    GP1:
        UF : 6, UT : 5,     CONFIG: 'N U T, 0, 0, 0',
       X = -410.7 mm, Y = 413.9 mm, Z = 598.9 mm,
       W = -11.9 deg, P = 9.7 deg,
    GP2:
        UF : 1, UT : 2,
       J1 = 0.0 deg, J2 = 0.0 deg
 };
P[387] {
    GP1:
        UF : 6, UT : 5,     CONFIG: 'N U T, 0, 0, 0',
 X = -393.7 mm, Y = 484.9 mm, Z = 598.9 mm,       W = -11.9 deg, P = 9.7 deg,
    GP2:
        UF : 1, UT : 2,
       J1 = 0.0 deg, J2 = 0.0 deg
 };
P[143] {
    GP1:
        UF : 6, UT : 5,     CONFIG: 'N U T, 0, 0, 0',
       X = -412.1 mm, Y = 415.1 mm, Z = 598.9 mm,
       W = -12.0 deg, P = 9.6 deg,
    GP2:
        UF : 1, UT : 2,
       J1 = 0.0 deg, J2 = 0.0 deg
 };
P[388] {
    GP1:
        UF : 6, UT : 5,     CONFIG: 'N U T, 0, 0, 0',
 X = -395.1 mm, Y = 486.1 mm, Z = 598.9 mm,       W = -12.0 deg, P = 9.6 deg,
    GP2:
        UF : 1, UT : 2,
       J1 = 0.0 deg, J2 = 0.0 deg
 };
P[144] {
    GP1:
        UF : 6, UT : 5,     CONFIG: 'N U T, 0, 0, 0',
       X = -413.0 mm, Y = 415.8 mm, Z = 598.9 mm,
       W = -11.9 deg, P = 9.6 deg,
    GP2:
        UF : 1, UT : 2,
       J1 = 0.0 deg, J2 = 0.0 deg
 };
P[389] {
    GP1:
        UF : 6, UT : 5,     CONFIG: 'N U T, 0, 0, 0',
 X = -396.0 mm, Y = 486.8 mm, Z = 598.9 mm,       W = -11.9 deg, P = 9.6 deg,
    GP2:
        UF : 1, UT : 2,
       J1 = 0.0 deg, J2 = 0.0 deg
 };
P[145] {
    GP1:
        UF : 6, UT : 5,     CONFIG: 'N U T, 0, 0, 0',
       X = -413.8 mm, Y = 416.5 mm, Z = 598.9 mm,
       W = -11.5 deg, P = 10.2 deg,
    GP2:
        UF : 1, UT : 2,
       J1 = 0.0 deg, J2 = 0.0 deg
 };
P[390] {
    GP1:
        UF : 6, UT : 5,     CONFIG: 'N U T, 0, 0, 0',
 X = -396.8 mm, Y = 487.5 mm, Z = 598.9 mm,       W = -11.5 deg, P = 10.2 deg,
    GP2:
        UF : 1, UT : 2,
       J1 = 0.0 deg, J2 = 0.0 deg
 };
P[146] {
    GP1:
        UF : 6, UT : 5,     CONFIG: 'N U T, 0, 0, 0',
       X = -414.8 mm, Y = 417.4 mm, Z = 598.9 mm,
       W = -11.4 deg, P = 10.5 deg,
    GP2:
        UF : 1, UT : 2,
       J1 = 0.0 deg, J2 = 0.0 deg
 };
P[391] {
    GP1:
        UF : 6, UT : 5,     CONFIG: 'N U T, 0, 0, 0',
 X = -397.8 mm, Y = 488.4 mm, Z = 598.9 mm,       W = -11.4 deg, P = 10.5 deg,
    GP2:
        UF : 1, UT : 2,
       J1 = 0.0 deg, J2 = 0.0 deg
 };
P[147] {
    GP1:
        UF : 6, UT : 5,     CONFIG: 'N U T, 0, 0, 0',
       X = -415.4 mm, Y = 417.9 mm, Z = 598.9 mm,
       W = -11.3 deg, P = 10.9 deg,
    GP2:
        UF : 1, UT : 2,
       J1 = 0.0 deg, J2 = 0.0 deg
 };
P[392] {
    GP1:
        UF : 6, UT : 5,     CONFIG: 'N U T, 0, 0, 0',
 X = -398.4 mm, Y = 488.9 mm, Z = 598.9 mm,       W = -11.3 deg, P = 10.9 deg,
    GP2:
        UF : 1, UT : 2,
       J1 = 0.0 deg, J2 = 0.0 deg
 };
P[148] {
    GP1:
        UF : 6, UT : 5,     CONFIG: 'N U T, 0, 0, 0',
       X = -415.8 mm, Y = 418.3 mm, Z = 598.9 mm,
       W = -10.8 deg, P = 11.6 deg,
    GP2:
        UF : 1, UT : 2,
       J1 = 0.0 deg, J2 = 0.0 deg
 };
P[393] {
    GP1:
        UF : 6, UT : 5,     CONFIG: 'N U T, 0, 0, 0',
 X = -398.8 mm, Y = 489.3 mm, Z = 598.9 mm,       W = -10.8 deg, P = 11.6 deg,
    GP2:
        UF : 1, UT : 2,
       J1 = 0.0 deg, J2 = 0.0 deg
 };
P[149] {
    GP1:
        UF : 6, UT : 5,     CONFIG: 'N U T, 0, 0, 0',
       X = -416.1 mm, Y = 418.7 mm, Z = 598.9 mm,
       W = -10.1 deg, P = 12.3 deg,
    GP2:
        UF : 1, UT : 2,
       J1 = 0.0 deg, J2 = 0.0 deg
 };
P[394] {
    GP1:
        UF : 6, UT : 5,     CONFIG: 'N U T, 0, 0, 0',
 X = -399.1 mm, Y = 489.7 mm, Z = 598.9 mm,       W = -10.1 deg, P = 12.3 deg,
    GP2:
        UF : 1, UT : 2,
       J1 = 0.0 deg, J2 = 0.0 deg
 };
P[150] {
    GP1:
        UF : 6, UT : 5,     CONFIG: 'N U T, 0, 0, 0',
       X = -416.8 mm, Y = 419.6 mm, Z = 598.9 mm,
       W = -9.7 deg, P = 12.7 deg,
    GP2:
        UF : 1, UT : 2,
       J1 = 0.0 deg, J2 = 0.0 deg
 };
P[395] {
    GP1:
        UF : 6, UT : 5,     CONFIG: 'N U T, 0, 0, 0',
 X = -399.8 mm, Y = 490.6 mm, Z = 598.9 mm,       W = -9.7 deg, P = 12.7 deg,
    GP2:
        UF : 1, UT : 2,
       J1 = 0.0 deg, J2 = 0.0 deg
 };
P[151] {
    GP1:
        UF : 6, UT : 5,     CONFIG: 'N U T, 0, 0, 0',
       X = -417.3 mm, Y = 420.2 mm, Z = 598.9 mm,
       W = -9.6 deg, P = 12.8 deg,
    GP2:
        UF : 1, UT : 2,
       J1 = 0.0 deg, J2 = 0.0 deg
 };
P[396] {
    GP1:
        UF : 6, UT : 5,     CONFIG: 'N U T, 0, 0, 0',
 X = -400.3 mm, Y = 491.2 mm, Z = 598.9 mm,       W = -9.6 deg, P = 12.8 deg,
    GP2:
        UF : 1, UT : 2,
       J1 = 0.0 deg, J2 = 0.0 deg
 };
P[152] {
    GP1:
        UF : 6, UT : 5,     CONFIG: 'N U T, 0, 0, 0',
       X = -417.9 mm, Y = 421.0 mm, Z = 598.9 mm,
       W = -8.6 deg, P = 13.4 deg,
    GP2:
        UF : 1, UT : 2,
       J1 = 0.0 deg, J2 = 0.0 deg
 };
P[397] {
    GP1:
        UF : 6, UT : 5,     CONFIG: 'N U T, 0, 0, 0',
 X = -400.9 mm, Y = 492.0 mm, Z = 598.9 mm,       W = -8.6 deg, P = 13.4 deg,
    GP2:
        UF : 1, UT : 2,
       J1 = 0.0 deg, J2 = 0.0 deg
 };
P[153] {
    GP1:
        UF : 6, UT : 5,     CONFIG: 'N U T, 0, 0, 0',
       X = -418.3 mm, Y = 421.8 mm, Z = 598.9 mm,
       W = -7.8 deg, P = 13.9 deg,
    GP2:
        UF : 1, UT : 2,
       J1 = 0.0 deg, J2 = 0.0 deg
 };
P[398] {
    GP1:
        UF : 6, UT : 5,     CONFIG: 'N U T, 0, 0, 0',
 X = -401.3 mm, Y = 492.8 mm, Z = 598.9 mm,       W = -7.8 deg, P = 13.9 deg,
    GP2:
        UF : 1, UT : 2,
       J1 = 0.0 deg, J2 = 0.0 deg
 };
P[154] {
    GP1:
        UF : 6, UT : 5,     CONFIG: 'N U T, 0, 0, 0',
       X = -418.8 mm, Y = 422.7 mm, Z = 598.9 mm,
       W = -7.5 deg, P = 13.9 deg,
    GP2:
        UF : 1, UT : 2,
       J1 = 0.0 deg, J2 = 0.0 deg
 };
P[399] {
    GP1:
        UF : 6, UT : 5,     CONFIG: 'N U T, 0, 0, 0',
 X = -401.8 mm, Y = 493.7 mm, Z = 598.9 mm,       W = -7.5 deg, P = 13.9 deg,
    GP2:
        UF : 1, UT : 2,
       J1 = 0.0 deg, J2 = 0.0 deg
 };
P[155] {
    GP1:
        UF : 6, UT : 5,     CONFIG: 'N U T, 0, 0, 0',
       X = -418.9 mm, Y = 423.0 mm, Z = 598.9 mm,
       W = -7.2 deg, P = 14.1 deg,
    GP2:
        UF : 1, UT : 2,
       J1 = 0.0 deg, J2 = 0.0 deg
 };
P[400] {
    GP1:
        UF : 6, UT : 5,     CONFIG: 'N U T, 0, 0, 0',
 X = -401.9 mm, Y = 494.0 mm, Z = 598.9 mm,       W = -7.2 deg, P = 14.1 deg,
    GP2:
        UF : 1, UT : 2,
       J1 = 0.0 deg, J2 = 0.0 deg
 };
P[156] {
    GP1:
        UF : 6, UT : 5,     CONFIG: 'N U T, 0, 0, 0',
       X = -419.0 mm, Y = 423.2 mm, Z = 598.9 mm,
       W = -6.9 deg, P = 14.2 deg,
    GP2:
        UF : 1, UT : 2,
       J1 = 0.0 deg, J2 = 0.0 deg
 };
P[401] {
    GP1:
        UF : 6, UT : 5,     CONFIG: 'N U T, 0, 0, 0',
 X = -402.0 mm, Y = 494.2 mm, Z = 598.9 mm,       W = -6.9 deg, P = 14.2 deg,
    GP2:
        UF : 1, UT : 2,
       J1 = 0.0 deg, J2 = 0.0 deg
 };
P[157] {
    GP1:
        UF : 6, UT : 5,     CONFIG: 'N U T, 0, 0, 0',
       X = -419.1 mm, Y = 423.4 mm, Z = 598.9 mm,
       W = -6.6 deg, P = 14.3 deg,
    GP2:
        UF : 1, UT : 2,
       J1 = 0.0 deg, J2 = 0.0 deg
 };
P[402] {
    GP1:
        UF : 6, UT : 5,     CONFIG: 'N U T, 0, 0, 0',
 X = -402.1 mm, Y = 494.4 mm, Z = 598.9 mm,       W = -6.6 deg, P = 14.3 deg,
    GP2:
        UF : 1, UT : 2,
       J1 = 0.0 deg, J2 = 0.0 deg
 };
P[158] {
    GP1:
        UF : 6, UT : 5,     CONFIG: 'N U T, 0, 0, 0',
       X = -419.3 mm, Y = 423.7 mm, Z = 598.9 mm,
       W = -6.3 deg, P = 14.4 deg,
    GP2:
        UF : 1, UT : 2,
       J1 = 0.0 deg, J2 = 0.0 deg
 };
P[403] {
    GP1:
        UF : 6, UT : 5,     CONFIG: 'N U T, 0, 0, 0',
 X = -402.3 mm, Y = 494.7 mm, Z = 598.9 mm,       W = -6.3 deg, P = 14.4 deg,
    GP2:
        UF : 1, UT : 2,
       J1 = 0.0 deg, J2 = 0.0 deg
 };
P[159] {
    GP1:
        UF : 6, UT : 5,     CONFIG: 'N U T, 0, 0, 0',
       X = -419.4 mm, Y = 424.0 mm, Z = 598.9 mm,
       W = -5.9 deg, P = 14.5 deg,
    GP2:
        UF : 1, UT : 2,
       J1 = 0.0 deg, J2 = 0.0 deg
 };
P[404] {
    GP1:
        UF : 6, UT : 5,     CONFIG: 'N U T, 0, 0, 0',
 X = -402.4 mm, Y = 495.0 mm, Z = 598.9 mm,       W = -5.9 deg, P = 14.5 deg,
    GP2:
        UF : 1, UT : 2,
       J1 = 0.0 deg, J2 = 0.0 deg
 };
P[160] {
    GP1:
        UF : 6, UT : 5,     CONFIG: 'N U T, 0, 0, 0',
       X = -419.5 mm, Y = 424.3 mm, Z = 598.9 mm,
       W = -5.6 deg, P = 14.5 deg,
    GP2:
        UF : 1, UT : 2,
       J1 = 0.0 deg, J2 = 0.0 deg
 };
P[405] {
    GP1:
        UF : 6, UT : 5,     CONFIG: 'N U T, 0, 0, 0',
 X = -402.5 mm, Y = 495.3 mm, Z = 598.9 mm,       W = -5.6 deg, P = 14.5 deg,
    GP2:
        UF : 1, UT : 2,
       J1 = 0.0 deg, J2 = 0.0 deg
 };
P[161] {
    GP1:
        UF : 6, UT : 5,     CONFIG: 'N U T, 0, 0, 0',
       X = -419.6 mm, Y = 424.6 mm, Z = 598.9 mm,
       W = -5.3 deg, P = 14.5 deg,
    GP2:
        UF : 1, UT : 2,
       J1 = 0.0 deg, J2 = 0.0 deg
 };
P[406] {
    GP1:
        UF : 6, UT : 5,     CONFIG: 'N U T, 0, 0, 0',
 X = -402.6 mm, Y = 495.6 mm, Z = 598.9 mm,       W = -5.3 deg, P = 14.5 deg,
    GP2:
        UF : 1, UT : 2,
       J1 = 0.0 deg, J2 = 0.0 deg
 };
P[162] {
    GP1:
        UF : 6, UT : 5,     CONFIG: 'N U T, 0, 0, 0',
       X = -419.7 mm, Y = 424.9 mm, Z = 598.9 mm,
       W = -4.9 deg, P = 14.6 deg,
    GP2:
        UF : 1, UT : 2,
       J1 = 0.0 deg, J2 = 0.0 deg
 };
P[407] {
    GP1:
        UF : 6, UT : 5,     CONFIG: 'N U T, 0, 0, 0',
 X = -402.7 mm, Y = 495.9 mm, Z = 598.9 mm,       W = -4.9 deg, P = 14.6 deg,
    GP2:
        UF : 1, UT : 2,
       J1 = 0.0 deg, J2 = 0.0 deg
 };
P[163] {
    GP1:
        UF : 6, UT : 5,     CONFIG: 'N U T, 0, 0, 0',
       X = -420.1 mm, Y = 426.4 mm, Z = 598.9 mm,
       W = -4.0 deg, P = 14.2 deg,
    GP2:
        UF : 1, UT : 2,
       J1 = 0.0 deg, J2 = 0.0 deg
 };
P[408] {
    GP1:
        UF : 6, UT : 5,     CONFIG: 'N U T, 0, 0, 0',
 X = -403.1 mm, Y = 497.4 mm, Z = 598.9 mm,       W = -4.0 deg, P = 14.2 deg,
    GP2:
        UF : 1, UT : 2,
       J1 = 0.0 deg, J2 = 0.0 deg
 };
P[164] {
    GP1:
        UF : 6, UT : 5,     CONFIG: 'N U T, 0, 0, 0',
       X = -420.2 mm, Y = 426.8 mm, Z = 598.9 mm,
       W = -3.4 deg, P = 14.2 deg,
    GP2:
        UF : 1, UT : 2,
       J1 = 0.0 deg, J2 = 0.0 deg
 };
P[409] {
    GP1:
        UF : 6, UT : 5,     CONFIG: 'N U T, 0, 0, 0',
 X = -403.2 mm, Y = 497.8 mm, Z = 598.9 mm,       W = -3.4 deg, P = 14.2 deg,
    GP2:
        UF : 1, UT : 2,
       J1 = 0.0 deg, J2 = 0.0 deg
 };
P[165] {
    GP1:
        UF : 6, UT : 5,     CONFIG: 'N U T, 0, 0, 0',
       X = -420.3 mm, Y = 427.0 mm, Z = 598.9 mm,
       W = -3.1 deg, P = 14.2 deg,
    GP2:
        UF : 1, UT : 2,
       J1 = 0.0 deg, J2 = 0.0 deg
 };
P[410] {
    GP1:
        UF : 6, UT : 5,     CONFIG: 'N U T, 0, 0, 0',
 X = -403.3 mm, Y = 498.0 mm, Z = 598.9 mm,       W = -3.1 deg, P = 14.2 deg,
    GP2:
        UF : 1, UT : 2,
       J1 = 0.0 deg, J2 = 0.0 deg
 };
P[166] {
    GP1:
        UF : 6, UT : 5,     CONFIG: 'N U T, 0, 0, 0',
       X = -420.4 mm, Y = 427.2 mm, Z = 598.9 mm,
       W = -2.8 deg, P = 14.2 deg,
    GP2:
        UF : 1, UT : 2,
       J1 = 0.0 deg, J2 = 0.0 deg
 };
P[411] {
    GP1:
        UF : 6, UT : 5,     CONFIG: 'N U T, 0, 0, 0',
 X = -403.4 mm, Y = 498.2 mm, Z = 598.9 mm,       W = -2.8 deg, P = 14.2 deg,
    GP2:
        UF : 1, UT : 2,
       J1 = 0.0 deg, J2 = 0.0 deg
 };
P[167] {
    GP1:
        UF : 6, UT : 5,     CONFIG: 'N U T, 0, 0, 0',
       X = -420.5 mm, Y = 428.0 mm, Z = 598.9 mm,
       W = -2.5 deg, P = 14.2 deg,
    GP2:
        UF : 1, UT : 2,
       J1 = 0.0 deg, J2 = 0.0 deg
 };
P[412] {
    GP1:
        UF : 6, UT : 5,     CONFIG: 'N U T, 0, 0, 0',
 X = -403.5 mm, Y = 499.0 mm, Z = 598.9 mm,       W = -2.5 deg, P = 14.2 deg,
    GP2:
        UF : 1, UT : 2,
       J1 = 0.0 deg, J2 = 0.0 deg
 };
P[168] {
    GP1:
        UF : 6, UT : 5,     CONFIG: 'N U T, 0, 0, 0',
       X = -420.7 mm, Y = 429.3 mm, Z = 598.9 mm,
       W = -1.5 deg, P = 14.1 deg,
    GP2:
        UF : 1, UT : 2,
       J1 = 0.0 deg, J2 = 0.0 deg
 };
P[413] {
    GP1:
        UF : 6, UT : 5,     CONFIG: 'N U T, 0, 0, 0',
 X = -403.7 mm, Y = 500.3 mm, Z = 598.9 mm,       W = -1.5 deg, P = 14.1 deg,
    GP2:
        UF : 1, UT : 2,
       J1 = 0.0 deg, J2 = 0.0 deg
 };
P[169] {
    GP1:
        UF : 6, UT : 5,     CONFIG: 'N U T, 0, 0, 0',
       X = -420.7 mm, Y = 429.7 mm, Z = 598.9 mm,
       W = -1.2 deg, P = 13.9 deg,
    GP2:
        UF : 1, UT : 2,
       J1 = 0.0 deg, J2 = 0.0 deg
 };
P[414] {
    GP1:
        UF : 6, UT : 5,     CONFIG: 'N U T, 0, 0, 0',
 X = -403.7 mm, Y = 500.7 mm, Z = 598.9 mm,       W = -1.2 deg, P = 13.9 deg,
    GP2:
        UF : 1, UT : 2,
       J1 = 0.0 deg, J2 = 0.0 deg
 };
P[170] {
    GP1:
        UF : 6, UT : 5,     CONFIG: 'N U T, 0, 0, 0',
       X = -420.7 mm, Y = 430.0 mm, Z = 598.9 mm,
       W = -0.8 deg, P = 13.6 deg,
    GP2:
        UF : 1, UT : 2,
       J1 = 0.0 deg, J2 = 0.0 deg
 };
P[415] {
    GP1:
        UF : 6, UT : 5,     CONFIG: 'N U T, 0, 0, 0',
 X = -403.7 mm, Y = 501.0 mm, Z = 598.9 mm,       W = -0.8 deg, P = 13.6 deg,
    GP2:
        UF : 1, UT : 2,
       J1 = 0.0 deg, J2 = 0.0 deg
 };
P[171] {
    GP1:
        UF : 6, UT : 5,     CONFIG: 'N U T, 0, 0, 0',
       X = -420.7 mm, Y = 430.4 mm, Z = 598.9 mm,
       W = -0.4 deg, P = 13.4 deg,
    GP2:
        UF : 1, UT : 2,
       J1 = 0.0 deg, J2 = 0.0 deg
 };
P[416] {
    GP1:
        UF : 6, UT : 5,     CONFIG: 'N U T, 0, 0, 0',
 X = -403.7 mm, Y = 501.4 mm, Z = 598.9 mm,       W = -0.4 deg, P = 13.4 deg,
    GP2:
        UF : 1, UT : 2,
       J1 = 0.0 deg, J2 = 0.0 deg
 };
P[172] {
    GP1:
        UF : 6, UT : 5,     CONFIG: 'N U T, 0, 0, 0',
       X = -420.7 mm, Y = 430.7 mm, Z = 598.9 mm,
       W = -0.1 deg, P = 13.2 deg,
    GP2:
        UF : 1, UT : 2,
       J1 = 0.0 deg, J2 = 0.0 deg
 };
P[417] {
    GP1:
        UF : 6, UT : 5,     CONFIG: 'N U T, 0, 0, 0',
 X = -403.7 mm, Y = 501.7 mm, Z = 598.9 mm,       W = -0.1 deg, P = 13.2 deg,
    GP2:
        UF : 1, UT : 2,
       J1 = 0.0 deg, J2 = 0.0 deg
 };
P[173] {
    GP1:
        UF : 6, UT : 5,     CONFIG: 'N U T, 0, 0, 0',
       X = -420.7 mm, Y = 432.1 mm, Z = 598.9 mm,
       W = 0.7 deg, P = 12.5 deg,
    GP2:
        UF : 1, UT : 2,
       J1 = 0.0 deg, J2 = 0.0 deg
 };
P[418] {
    GP1:
        UF : 6, UT : 5,     CONFIG: 'N U T, 0, 0, 0',
 X = -403.7 mm, Y = 503.1 mm, Z = 598.9 mm,       W = 0.7 deg, P = 12.5 deg,
    GP2:
        UF : 1, UT : 2,
       J1 = 0.0 deg, J2 = 0.0 deg
 };
P[174] {
    GP1:
        UF : 6, UT : 5,     CONFIG: 'N U T, 0, 0, 0',
       X = -420.7 mm, Y = 432.4 mm, Z = 598.9 mm,
       W = 0.9 deg, P = 12.3 deg,
    GP2:
        UF : 1, UT : 2,
       J1 = 0.0 deg, J2 = 0.0 deg
 };
P[419] {
    GP1:
        UF : 6, UT : 5,     CONFIG: 'N U T, 0, 0, 0',
 X = -403.7 mm, Y = 503.4 mm, Z = 598.9 mm,       W = 0.9 deg, P = 12.3 deg,
    GP2:
        UF : 1, UT : 2,
       J1 = 0.0 deg, J2 = 0.0 deg
 };
P[175] {
    GP1:
        UF : 6, UT : 5,     CONFIG: 'N U T, 0, 0, 0',
       X = -420.7 mm, Y = 432.7 mm, Z = 598.9 mm,
       W = 1.2 deg, P = 12.0 deg,
    GP2:
        UF : 1, UT : 2,
       J1 = 0.0 deg, J2 = 0.0 deg
 };
P[420] {
    GP1:
        UF : 6, UT : 5,     CONFIG: 'N U T, 0, 0, 0',
 X = -403.7 mm, Y = 503.7 mm, Z = 598.9 mm,       W = 1.2 deg, P = 12.0 deg,
    GP2:
        UF : 1, UT : 2,
       J1 = 0.0 deg, J2 = 0.0 deg
 };
P[176] {
    GP1:
        UF : 6, UT : 5,     CONFIG: 'N U T, 0, 0, 0',
       X = -420.6 mm, Y = 433.0 mm, Z = 598.9 mm,
       W = 1.4 deg, P = 11.8 deg,
    GP2:
        UF : 1, UT : 2,
       J1 = 0.0 deg, J2 = 0.0 deg
 };
P[421] {
    GP1:
        UF : 6, UT : 5,     CONFIG: 'N U T, 0, 0, 0',
 X = -403.6 mm, Y = 504.0 mm, Z = 598.9 mm,       W = 1.4 deg, P = 11.8 deg,
    GP2:
        UF : 1, UT : 2,
       J1 = 0.0 deg, J2 = 0.0 deg
 };
P[177] {
    GP1:
        UF : 6, UT : 5,     CONFIG: 'N U T, 0, 0, 0',
       X = -420.6 mm, Y = 433.4 mm, Z = 598.9 mm,
       W = 1.7 deg, P = 11.5 deg,
    GP2:
        UF : 1, UT : 2,
       J1 = 0.0 deg, J2 = 0.0 deg
 };
P[422] {
    GP1:
        UF : 6, UT : 5,     CONFIG: 'N U T, 0, 0, 0',
 X = -403.6 mm, Y = 504.4 mm, Z = 598.9 mm,       W = 1.7 deg, P = 11.5 deg,
    GP2:
        UF : 1, UT : 2,
       J1 = 0.0 deg, J2 = 0.0 deg
 };
P[178] {
    GP1:
        UF : 6, UT : 5,     CONFIG: 'N U T, 0, 0, 0',
       X = -420.3 mm, Y = 434.9 mm, Z = 598.9 mm,
       W = 2.3 deg, P = 11.3 deg,
    GP2:
        UF : 1, UT : 2,
       J1 = 0.0 deg, J2 = 0.0 deg
 };
P[423] {
    GP1:
        UF : 6, UT : 5,     CONFIG: 'N U T, 0, 0, 0',
 X = -403.3 mm, Y = 505.9 mm, Z = 598.9 mm,       W = 2.3 deg, P = 11.3 deg,
    GP2:
        UF : 1, UT : 2,
       J1 = 0.0 deg, J2 = 0.0 deg
 };
P[179] {
    GP1:
        UF : 6, UT : 5,     CONFIG: 'N U T, 0, 0, 0',
       X = -420.1 mm, Y = 435.7 mm, Z = 598.9 mm,
       W = 3.0 deg, P = 10.9 deg,
    GP2:
        UF : 1, UT : 2,
       J1 = 0.0 deg, J2 = 0.0 deg
 };
P[424] {
    GP1:
        UF : 6, UT : 5,     CONFIG: 'N U T, 0, 0, 0',
 X = -403.1 mm, Y = 506.7 mm, Z = 598.9 mm,       W = 3.0 deg, P = 10.9 deg,
    GP2:
        UF : 1, UT : 2,
       J1 = 0.0 deg, J2 = 0.0 deg
 };
P[180] {
    GP1:
        UF : 6, UT : 5,     CONFIG: 'N U T, 0, 0, 0',
       X = -419.9 mm, Y = 436.5 mm, Z = 598.9 mm,
       W = 3.4 deg, P = 9.7 deg,
    GP2:
        UF : 1, UT : 2,
       J1 = 0.0 deg, J2 = 0.0 deg
 };
P[425] {
    GP1:
        UF : 6, UT : 5,     CONFIG: 'N U T, 0, 0, 0',
 X = -402.9 mm, Y = 507.5 mm, Z = 598.9 mm,       W = 3.4 deg, P = 9.7 deg,
    GP2:
        UF : 1, UT : 2,
       J1 = 0.0 deg, J2 = 0.0 deg
 };
P[181] {
    GP1:
        UF : 6, UT : 5,     CONFIG: 'N U T, 0, 0, 0',
       X = -419.6 mm, Y = 437.3 mm, Z = 598.9 mm,
       W = 3.3 deg, P = 9.1 deg,
    GP2:
        UF : 1, UT : 2,
       J1 = 0.0 deg, J2 = 0.0 deg
 };
P[426] {
    GP1:
        UF : 6, UT : 5,     CONFIG: 'N U T, 0, 0, 0',
 X = -402.6 mm, Y = 508.3 mm, Z = 598.9 mm,       W = 3.3 deg, P = 9.1 deg,
    GP2:
        UF : 1, UT : 2,
       J1 = 0.0 deg, J2 = 0.0 deg
 };
P[182] {
    GP1:
        UF : 6, UT : 5,     CONFIG: 'N U T, 0, 0, 0',
       X = -419.2 mm, Y = 438.2 mm, Z = 598.9 mm,
       W = 3.7 deg, P = 8.7 deg,
    GP2:
        UF : 1, UT : 2,
       J1 = 0.0 deg, J2 = 0.0 deg
 };
P[427] {
    GP1:
        UF : 6, UT : 5,     CONFIG: 'N U T, 0, 0, 0',
 X = -402.2 mm, Y = 509.2 mm, Z = 598.9 mm,       W = 3.7 deg, P = 8.7 deg,
    GP2:
        UF : 1, UT : 2,
       J1 = 0.0 deg, J2 = 0.0 deg
 };
P[183] {
    GP1:
        UF : 6, UT : 5,     CONFIG: 'N U T, 0, 0, 0',
       X = -419.1 mm, Y = 438.5 mm, Z = 598.9 mm,
       W = 3.8 deg, P = 8.4 deg,
    GP2:
        UF : 1, UT : 2,
       J1 = 0.0 deg, J2 = 0.0 deg
 };
P[428] {
    GP1:
        UF : 6, UT : 5,     CONFIG: 'N U T, 0, 0, 0',
 X = -402.1 mm, Y = 509.5 mm, Z = 598.9 mm,       W = 3.8 deg, P = 8.4 deg,
    GP2:
        UF : 1, UT : 2,
       J1 = 0.0 deg, J2 = 0.0 deg
 };
P[184] {
    GP1:
        UF : 6, UT : 5,     CONFIG: 'N U T, 0, 0, 0',
       X = -419.0 mm, Y = 438.7 mm, Z = 598.9 mm,
       W = 3.8 deg, P = 8.1 deg,
    GP2:
        UF : 1, UT : 2,
       J1 = 0.0 deg, J2 = 0.0 deg
 };
P[429] {
    GP1:
        UF : 6, UT : 5,     CONFIG: 'N U T, 0, 0, 0',
 X = -402.0 mm, Y = 509.7 mm, Z = 598.9 mm,       W = 3.8 deg, P = 8.1 deg,
    GP2:
        UF : 1, UT : 2,
       J1 = 0.0 deg, J2 = 0.0 deg
 };
P[185] {
    GP1:
        UF : 6, UT : 5,     CONFIG: 'N U T, 0, 0, 0',
       X = -418.9 mm, Y = 438.9 mm, Z = 598.9 mm,
       W = 3.9 deg, P = 7.9 deg,
    GP2:
        UF : 1, UT : 2,
       J1 = 0.0 deg, J2 = 0.0 deg
 };
P[430] {
    GP1:
        UF : 6, UT : 5,     CONFIG: 'N U T, 0, 0, 0',
 X = -401.9 mm, Y = 509.9 mm, Z = 598.9 mm,       W = 3.9 deg, P = 7.9 deg,
    GP2:
        UF : 1, UT : 2,
       J1 = 0.0 deg, J2 = 0.0 deg
 };
P[186] {
    GP1:
        UF : 6, UT : 5,     CONFIG: 'N U T, 0, 0, 0',
       X = -418.8 mm, Y = 439.2 mm, Z = 598.9 mm,
       W = 4.0 deg, P = 7.6 deg,
    GP2:
        UF : 1, UT : 2,
       J1 = 0.0 deg, J2 = 0.0 deg
 };
P[431] {
    GP1:
        UF : 6, UT : 5,     CONFIG: 'N U T, 0, 0, 0',
 X = -401.8 mm, Y = 510.2 mm, Z = 598.9 mm,       W = 4.0 deg, P = 7.6 deg,
    GP2:
        UF : 1, UT : 2,
       J1 = 0.0 deg, J2 = 0.0 deg
 };
P[187] {
    GP1:
        UF : 6, UT : 5,     CONFIG: 'N U T, 0, 0, 0',
       X = -418.1 mm, Y = 440.5 mm, Z = 598.9 mm,
       W = 3.5 deg, P = 6.0 deg,
    GP2:
        UF : 1, UT : 2,
       J1 = 0.0 deg, J2 = 0.0 deg
 };
P[432] {
    GP1:
        UF : 6, UT : 5,     CONFIG: 'N U T, 0, 0, 0',
 X = -401.1 mm, Y = 511.5 mm, Z = 598.9 mm,       W = 3.5 deg, P = 6.0 deg,
    GP2:
        UF : 1, UT : 2,
       J1 = 0.0 deg, J2 = 0.0 deg
 };
P[188] {
    GP1:
        UF : 6, UT : 5,     CONFIG: 'N U T, 0, 0, 0',
       X = -417.6 mm, Y = 441.3 mm, Z = 598.9 mm,
       W = 3.5 deg, P = 5.3 deg,
    GP2:
        UF : 1, UT : 2,
       J1 = 0.0 deg, J2 = 0.0 deg
 };
P[433] {
    GP1:
        UF : 6, UT : 5,     CONFIG: 'N U T, 0, 0, 0',
 X = -400.6 mm, Y = 512.3 mm, Z = 598.9 mm,       W = 3.5 deg, P = 5.3 deg,
    GP2:
        UF : 1, UT : 2,
       J1 = 0.0 deg, J2 = 0.0 deg
 };
P[189] {
    GP1:
        UF : 6, UT : 5,     CONFIG: 'N U T, 0, 0, 0',
       X = -417.5 mm, Y = 441.4 mm, Z = 598.9 mm,
       W = 3.5 deg, P = 5.1 deg,
    GP2:
        UF : 1, UT : 2,
       J1 = 0.0 deg, J2 = 0.0 deg
 };
P[434] {
    GP1:
        UF : 6, UT : 5,     CONFIG: 'N U T, 0, 0, 0',
 X = -400.5 mm, Y = 512.4 mm, Z = 598.9 mm,       W = 3.5 deg, P = 5.1 deg,
    GP2:
        UF : 1, UT : 2,
       J1 = 0.0 deg, J2 = 0.0 deg
 };
P[190] {
    GP1:
        UF : 6, UT : 5,     CONFIG: 'N U T, 0, 0, 0',
       X = -417.4 mm, Y = 441.6 mm, Z = 598.9 mm,
       W = 3.5 deg, P = 4.9 deg,
    GP2:
        UF : 1, UT : 2,
       J1 = 0.0 deg, J2 = 0.0 deg
 };
P[435] {
    GP1:
        UF : 6, UT : 5,     CONFIG: 'N U T, 0, 0, 0',
 X = -400.4 mm, Y = 512.6 mm, Z = 598.9 mm,       W = 3.5 deg, P = 4.9 deg,
    GP2:
        UF : 1, UT : 2,
       J1 = 0.0 deg, J2 = 0.0 deg
 };
P[191] {
    GP1:
        UF : 6, UT : 5,     CONFIG: 'N U T, 0, 0, 0',
       X = -417.3 mm, Y = 441.7 mm, Z = 598.9 mm,
       W = 3.5 deg, P = 4.8 deg,
    GP2:
        UF : 1, UT : 2,
       J1 = 0.0 deg, J2 = 0.0 deg
 };
P[436] {
    GP1:
        UF : 6, UT : 5,     CONFIG: 'N U T, 0, 0, 0',
 X = -400.3 mm, Y = 512.7 mm, Z = 598.9 mm,       W = 3.5 deg, P = 4.8 deg,
    GP2:
        UF : 1, UT : 2,
       J1 = 0.0 deg, J2 = 0.0 deg
 };
P[192] {
    GP1:
        UF : 6, UT : 5,     CONFIG: 'N U T, 0, 0, 0',
       X = -417.1 mm, Y = 441.9 mm, Z = 598.9 mm,
       W = 3.5 deg, P = 4.5 deg,
    GP2:
        UF : 1, UT : 2,
       J1 = 0.0 deg, J2 = 0.0 deg
 };
P[437] {
    GP1:
        UF : 6, UT : 5,     CONFIG: 'N U T, 0, 0, 0',
 X = -400.1 mm, Y = 512.9 mm, Z = 598.9 mm,       W = 3.5 deg, P = 4.5 deg,
    GP2:
        UF : 1, UT : 2,
       J1 = 0.0 deg, J2 = 0.0 deg
 };
P[193] {
    GP1:
        UF : 6, UT : 5,     CONFIG: 'N U T, 0, 0, 0',
       X = -416.6 mm, Y = 442.6 mm, Z = 598.9 mm,
       W = 3.2 deg, P = 4.0 deg,
    GP2:
        UF : 1, UT : 2,
       J1 = 0.0 deg, J2 = 0.0 deg
 };
P[438] {
    GP1:
        UF : 6, UT : 5,     CONFIG: 'N U T, 0, 0, 0',
 X = -399.6 mm, Y = 513.6 mm, Z = 598.9 mm,       W = 3.2 deg, P = 4.0 deg,
    GP2:
        UF : 1, UT : 2,
       J1 = 0.0 deg, J2 = 0.0 deg
 };
P[194] {
    GP1:
        UF : 6, UT : 5,     CONFIG: 'N U T, 0, 0, 0',
       X = -414.6 mm, Y = 444.9 mm, Z = 598.9 mm,
       W = 2.9 deg, P = 3.4 deg,
    GP2:
        UF : 1, UT : 2,
       J1 = 0.0 deg, J2 = 0.0 deg
 };
P[439] {
    GP1:
        UF : 6, UT : 5,     CONFIG: 'N U T, 0, 0, 0',
 X = -397.6 mm, Y = 515.9 mm, Z = 598.9 mm,       W = 2.9 deg, P = 3.4 deg,
    GP2:
        UF : 1, UT : 2,
       J1 = 0.0 deg, J2 = 0.0 deg
 };
P[195] {
    GP1:
        UF : 6, UT : 5,     CONFIG: 'N U T, 0, 0, 0',
       X = -407.9 mm, Y = 451.9 mm, Z = 598.9 mm,
       W = 2.8 deg, P = 3.2 deg,
    GP2:
        UF : 1, UT : 2,
       J1 = 0.0 deg, J2 = 0.0 deg
 };
P[440] {
    GP1:
        UF : 6, UT : 5,     CONFIG: 'N U T, 0, 0, 0',
 X = -390.9 mm, Y = 522.9 mm, Z = 598.9 mm,       W = 2.8 deg, P = 3.2 deg,
    GP2:
        UF : 1, UT : 2,
       J1 = 0.0 deg, J2 = 0.0 deg
 };
P[196] {
    GP1:
        UF : 6, UT : 5,     CONFIG: 'N U T, 0, 0, 0',
       X = -401.2 mm, Y = 458.8 mm, Z = 598.9 mm,
       W = 2.6 deg, P = 3.0 deg,
    GP2:
        UF : 1, UT : 2,
       J1 = 0.0 deg, J2 = 0.0 deg
 };
P[441] {
    GP1:
        UF : 6, UT : 5,     CONFIG: 'N U T, 0, 0, 0',
 X = -384.2 mm, Y = 529.8 mm, Z = 598.9 mm,       W = 2.6 deg, P = 3.0 deg,
    GP2:
        UF : 1, UT : 2,
       J1 = 0.0 deg, J2 = 0.0 deg
 };
P[197] {
    GP1:
        UF : 6, UT : 5,     CONFIG: 'N U T, 0, 0, 0',
       X = -394.3 mm, Y = 465.6 mm, Z = 598.9 mm,
       W = 2.4 deg, P = 2.8 deg,
    GP2:
        UF : 1, UT : 2,
       J1 = 0.0 deg, J2 = 0.0 deg
 };
P[442] {
    GP1:
        UF : 6, UT : 5,     CONFIG: 'N U T, 0, 0, 0',
 X = -377.3 mm, Y = 536.6 mm, Z = 598.9 mm,       W = 2.4 deg, P = 2.8 deg,
    GP2:
        UF : 1, UT : 2,
       J1 = 0.0 deg, J2 = 0.0 deg
 };
P[198] {
    GP1:
        UF : 6, UT : 5,     CONFIG: 'N U T, 0, 0, 0',
       X = -387.4 mm, Y = 472.3 mm, Z = 598.9 mm,
       W = 2.2 deg, P = 2.6 deg,
    GP2:
        UF : 1, UT : 2,
       J1 = 0.0 deg, J2 = 0.0 deg
 };
P[443] {
    GP1:
        UF : 6, UT : 5,     CONFIG: 'N U T, 0, 0, 0',
 X = -370.4 mm, Y = 543.3 mm, Z = 598.9 mm,       W = 2.2 deg, P = 2.6 deg,
    GP2:
        UF : 1, UT : 2,
       J1 = 0.0 deg, J2 = 0.0 deg
 };
P[199] {
    GP1:
        UF : 6, UT : 5,     CONFIG: 'N U T, 0, 0, 0',
       X = -383.7 mm, Y = 475.8 mm, Z = 598.9 mm,
       W = 2.1 deg, P = 2.5 deg,
    GP2:
        UF : 1, UT : 2,
       J1 = 0.0 deg, J2 = 0.0 deg
 };
P[444] {
    GP1:
        UF : 6, UT : 5,     CONFIG: 'N U T, 0, 0, 0',
 X = -366.7 mm, Y = 546.8 mm, Z = 598.9 mm,       W = 2.1 deg, P = 2.5 deg,
    GP2:
        UF : 1, UT : 2,
       J1 = 0.0 deg, J2 = 0.0 deg
 };
P[200] {
    GP1:
        UF : 6, UT : 5,     CONFIG: 'N U T, 0, 0, 0',
       X = -382.4 mm, Y = 477.2 mm, Z = 598.9 mm,
       W = 2.1 deg, P = 2.5 deg,
    GP2:
        UF : 1, UT : 2,
       J1 = 0.0 deg, J2 = 0.0 deg
 };
P[445] {
    GP1:
        UF : 6, UT : 5,     CONFIG: 'N U T, 0, 0, 0',
 X = -365.4 mm, Y = 548.2 mm, Z = 598.9 mm,       W = 2.1 deg, P = 2.5 deg,
    GP2:
        UF : 1, UT : 2,
       J1 = 0.0 deg, J2 = 0.0 deg
 };
P[201] {
    GP1:
        UF : 6, UT : 5,     CONFIG: 'N U T, 0, 0, 0',
       X = -381.1 mm, Y = 478.6 mm, Z = 598.9 mm,
       W = 2.1 deg, P = 2.4 deg,
    GP2:
        UF : 1, UT : 2,
       J1 = 0.0 deg, J2 = 0.0 deg
 };
P[446] {
    GP1:
        UF : 6, UT : 5,     CONFIG: 'N U T, 0, 0, 0',
 X = -364.1 mm, Y = 549.6 mm, Z = 598.9 mm,       W = 2.1 deg, P = 2.4 deg,
    GP2:
        UF : 1, UT : 2,
       J1 = 0.0 deg, J2 = 0.0 deg
 };
P[202] {
    GP1:
        UF : 6, UT : 5,     CONFIG: 'N U T, 0, 0, 0',
       X = -380.3 mm, Y = 479.6 mm, Z = 598.9 mm,
       W = 2.0 deg, P = 2.4 deg,
    GP2:
        UF : 1, UT : 2,
       J1 = 0.0 deg, J2 = 0.0 deg
 };
P[447] {
    GP1:
        UF : 6, UT : 5,     CONFIG: 'N U T, 0, 0, 0',
 X = -363.3 mm, Y = 550.6 mm, Z = 598.9 mm,       W = 2.0 deg, P = 2.4 deg,
    GP2:
        UF : 1, UT : 2,
       J1 = 0.0 deg, J2 = 0.0 deg
 };
P[203] {
    GP1:
        UF : 6, UT : 5,     CONFIG: 'N U T, 0, 0, 0',
       X = -379.7 mm, Y = 480.8 mm, Z = 598.9 mm,
       W = 2.0 deg, P = 2.4 deg,
    GP2:
        UF : 1, UT : 2,
       J1 = 0.0 deg, J2 = 0.0 deg
 };
P[448] {
    GP1:
        UF : 6, UT : 5,     CONFIG: 'N U T, 0, 0, 0',
 X = -362.7 mm, Y = 551.8 mm, Z = 598.9 mm,       W = 2.0 deg, P = 2.4 deg,
    GP2:
        UF : 1, UT : 2,
       J1 = 0.0 deg, J2 = 0.0 deg
 };
P[204] {
    GP1:
        UF : 6, UT : 5,     CONFIG: 'N U T, 0, 0, 0',
       X = -379.2 mm, Y = 482.0 mm, Z = 598.9 mm,
       W = 1.9 deg, P = 2.4 deg,
    GP2:
        UF : 1, UT : 2,
       J1 = 0.0 deg, J2 = 0.0 deg
 };
P[449] {
    GP1:
        UF : 6, UT : 5,     CONFIG: 'N U T, 0, 0, 0',
 X = -362.2 mm, Y = 553.0 mm, Z = 598.9 mm,       W = 1.9 deg, P = 2.4 deg,
    GP2:
        UF : 1, UT : 2,
       J1 = 0.0 deg, J2 = 0.0 deg
 };
P[205] {
    GP1:
        UF : 6, UT : 5,     CONFIG: 'N U T, 0, 0, 0',
       X = -378.7 mm, Y = 484.0 mm, Z = 598.9 mm,
       W = 1.9 deg, P = 2.3 deg,
    GP2:
        UF : 1, UT : 2,
       J1 = 0.0 deg, J2 = 0.0 deg
 };
P[450] {
    GP1:
        UF : 6, UT : 5,     CONFIG: 'N U T, 0, 0, 0',
 X = -361.7 mm, Y = 555.0 mm, Z = 598.9 mm,       W = 1.9 deg, P = 2.3 deg,
    GP2:
        UF : 1, UT : 2,
       J1 = 0.0 deg, J2 = 0.0 deg
 };
P[206] {
    GP1:
        UF : 6, UT : 5,     CONFIG: 'N U T, 0, 0, 0',
       X = -378.5 mm, Y = 486.3 mm, Z = 598.9 mm,
       W = 1.9 deg, P = 2.2 deg,
    GP2:
        UF : 1, UT : 2,
       J1 = 0.0 deg, J2 = 0.0 deg
 };
P[451] {
    GP1:
        UF : 6, UT : 5,     CONFIG: 'N U T, 0, 0, 0',
 X = -361.5 mm, Y = 557.3 mm, Z = 598.9 mm,       W = 1.9 deg, P = 2.2 deg,
    GP2:
        UF : 1, UT : 2,
       J1 = 0.0 deg, J2 = 0.0 deg
 };
P[207] {
    GP1:
        UF : 6, UT : 5,     CONFIG: 'N U T, 0, 0, 0',
       X = -378.7 mm, Y = 488.4 mm, Z = 598.9 mm,
       W = 1.8 deg, P = 2.2 deg,
    GP2:
        UF : 1, UT : 2,
       J1 = 0.0 deg, J2 = 0.0 deg
 };
P[452] {
    GP1:
        UF : 6, UT : 5,     CONFIG: 'N U T, 0, 0, 0',
 X = -361.7 mm, Y = 559.4 mm, Z = 598.9 mm,       W = 1.8 deg, P = 2.2 deg,
    GP2:
        UF : 1, UT : 2,
       J1 = 0.0 deg, J2 = 0.0 deg
 };
P[208] {
    GP1:
        UF : 6, UT : 5,     CONFIG: 'N U T, 0, 0, 0',
       X = -379.4 mm, Y = 490.6 mm, Z = 598.9 mm,
       W = 1.8 deg, P = 2.1 deg,
    GP2:
        UF : 1, UT : 2,
       J1 = 0.0 deg, J2 = 0.0 deg
 };
P[453] {
    GP1:
        UF : 6, UT : 5,     CONFIG: 'N U T, 0, 0, 0',
 X = -362.4 mm, Y = 561.6 mm, Z = 598.9 mm,       W = 1.8 deg, P = 2.1 deg,
    GP2:
        UF : 1, UT : 2,
       J1 = 0.0 deg, J2 = 0.0 deg
 };
P[209] {
    GP1:
        UF : 6, UT : 5,     CONFIG: 'N U T, 0, 0, 0',
       X = -380.0 mm, Y = 491.8 mm, Z = 598.9 mm,
       W = 1.8 deg, P = 2.1 deg,
    GP2:
        UF : 1, UT : 2,
       J1 = 0.0 deg, J2 = 0.0 deg
 };
P[454] {
    GP1:
        UF : 6, UT : 5,     CONFIG: 'N U T, 0, 0, 0',
 X = -363.0 mm, Y = 562.8 mm, Z = 598.9 mm,       W = 1.8 deg, P = 2.1 deg,
    GP2:
        UF : 1, UT : 2,
       J1 = 0.0 deg, J2 = 0.0 deg
 };
P[210] {
    GP1:
        UF : 6, UT : 5,     CONFIG: 'N U T, 0, 0, 0',
       X = -380.9 mm, Y = 492.9 mm, Z = 598.9 mm,
       W = 1.8 deg, P = 2.1 deg,
    GP2:
        UF : 1, UT : 2,
       J1 = 0.0 deg, J2 = 0.0 deg
 };
P[455] {
    GP1:
        UF : 6, UT : 5,     CONFIG: 'N U T, 0, 0, 0',
 X = -363.9 mm, Y = 563.9 mm, Z = 598.9 mm,       W = 1.8 deg, P = 2.1 deg,
    GP2:
        UF : 1, UT : 2,
       J1 = 0.0 deg, J2 = 0.0 deg
 };
P[211] {
    GP1:
        UF : 6, UT : 5,     CONFIG: 'N U T, 0, 0, 0',
       X = -382.0 mm, Y = 494.0 mm, Z = 598.9 mm,
       W = 1.7 deg, P = 2.1 deg,
    GP2:
        UF : 1, UT : 2,
       J1 = 0.0 deg, J2 = 0.0 deg
 };
P[456] {
    GP1:
        UF : 6, UT : 5,     CONFIG: 'N U T, 0, 0, 0',
 X = -365.0 mm, Y = 565.0 mm, Z = 598.9 mm,       W = 1.7 deg, P = 2.1 deg,
    GP2:
        UF : 1, UT : 2,
       J1 = 0.0 deg, J2 = 0.0 deg
 };
P[212] {
    GP1:
        UF : 6, UT : 5,     CONFIG: 'N U T, 0, 0, 0',
       X = -384.2 mm, Y = 495.8 mm, Z = 598.9 mm,
       W = 1.7 deg, P = 2.0 deg,
    GP2:
        UF : 1, UT : 2,
       J1 = 0.0 deg, J2 = 0.0 deg
 };
P[457] {
    GP1:
        UF : 6, UT : 5,     CONFIG: 'N U T, 0, 0, 0',
 X = -367.2 mm, Y = 566.8 mm, Z = 598.9 mm,       W = 1.7 deg, P = 2.0 deg,
    GP2:
        UF : 1, UT : 2,
       J1 = 0.0 deg, J2 = 0.0 deg
 };
P[213] {
    GP1:
        UF : 6, UT : 5,     CONFIG: 'N U T, 0, 0, 0',
       X = -392.3 mm, Y = 501.0 mm, Z = 598.9 mm,
       W = 1.5 deg, P = 1.8 deg,
    GP2:
        UF : 1, UT : 2,
       J1 = 0.0 deg, J2 = 0.0 deg
 };
P[458] {
    GP1:
        UF : 6, UT : 5,     CONFIG: 'N U T, 0, 0, 0',
 X = -375.3 mm, Y = 572.0 mm, Z = 598.9 mm,       W = 1.5 deg, P = 1.8 deg,
    GP2:
        UF : 1, UT : 2,
       J1 = 0.0 deg, J2 = 0.0 deg
 };
P[214] {
    GP1:
        UF : 6, UT : 5,     CONFIG: 'N U T, 0, 0, 0',
       X = -400.5 mm, Y = 506.1 mm, Z = 598.9 mm,
       W = 1.3 deg, P = 1.5 deg,
    GP2:
        UF : 1, UT : 2,
       J1 = 0.0 deg, J2 = 0.0 deg
 };
P[459] {
    GP1:
        UF : 6, UT : 5,     CONFIG: 'N U T, 0, 0, 0',
 X = -383.5 mm, Y = 577.1 mm, Z = 598.9 mm,       W = 1.3 deg, P = 1.5 deg,
    GP2:
        UF : 1, UT : 2,
       J1 = 0.0 deg, J2 = 0.0 deg
 };
P[215] {
    GP1:
        UF : 6, UT : 5,     CONFIG: 'N U T, 0, 0, 0',
       X = -408.8 mm, Y = 511.0 mm, Z = 598.9 mm,
       W = 1.1 deg, P = 1.3 deg,
    GP2:
        UF : 1, UT : 2,
       J1 = 0.0 deg, J2 = 0.0 deg
 };
P[460] {
    GP1:
        UF : 6, UT : 5,     CONFIG: 'N U T, 0, 0, 0',
 X = -391.8 mm, Y = 582.0 mm, Z = 598.9 mm,       W = 1.1 deg, P = 1.3 deg,
    GP2:
        UF : 1, UT : 2,
       J1 = 0.0 deg, J2 = 0.0 deg
 };
P[216] {
    GP1:
        UF : 6, UT : 5,     CONFIG: 'N U T, 0, 0, 0',
       X = -417.2 mm, Y = 515.8 mm, Z = 598.9 mm,
       W = 1.0 deg, P = 1.1 deg,
    GP2:
        UF : 1, UT : 2,
       J1 = 0.0 deg, J2 = 0.0 deg
 };
P[461] {
    GP1:
        UF : 6, UT : 5,     CONFIG: 'N U T, 0, 0, 0',
 X = -400.2 mm, Y = 586.8 mm, Z = 598.9 mm,       W = 1.0 deg, P = 1.1 deg,
    GP2:
        UF : 1, UT : 2,
       J1 = 0.0 deg, J2 = 0.0 deg
 };
P[217] {
    GP1:
        UF : 6, UT : 5,     CONFIG: 'N U T, 0, 0, 0',
       X = -425.6 mm, Y = 520.4 mm, Z = 598.9 mm,
       W = 0.8 deg, P = 0.9 deg,
    GP2:
        UF : 1, UT : 2,
       J1 = 0.0 deg, J2 = 0.0 deg
 };
P[462] {
    GP1:
        UF : 6, UT : 5,     CONFIG: 'N U T, 0, 0, 0',
 X = -408.6 mm, Y = 591.4 mm, Z = 598.9 mm,       W = 0.8 deg, P = 0.9 deg,
    GP2:
        UF : 1, UT : 2,
       J1 = 0.0 deg, J2 = 0.0 deg
 };
P[218] {
    GP1:
        UF : 6, UT : 5,     CONFIG: 'N U T, 0, 0, 0',
       X = -434.2 mm, Y = 524.9 mm, Z = 598.9 mm,
       W = 0.6 deg, P = 0.7 deg,
    GP2:
        UF : 1, UT : 2,
       J1 = 0.0 deg, J2 = 0.0 deg
 };
P[463] {
    GP1:
        UF : 6, UT : 5,     CONFIG: 'N U T, 0, 0, 0',
 X = -417.2 mm, Y = 595.9 mm, Z = 598.9 mm,       W = 0.6 deg, P = 0.7 deg,
    GP2:
        UF : 1, UT : 2,
       J1 = 0.0 deg, J2 = 0.0 deg
 };
P[219] {
    GP1:
        UF : 6, UT : 5,     CONFIG: 'N U T, 0, 0, 0',
       X = -439.8 mm, Y = 527.8 mm, Z = 598.9 mm,
       W = 0.5 deg, P = 0.6 deg,
    GP2:
        UF : 1, UT : 2,
       J1 = 0.0 deg, J2 = 0.0 deg
 };
P[464] {
    GP1:
        UF : 6, UT : 5,     CONFIG: 'N U T, 0, 0, 0',
 X = -422.8 mm, Y = 598.8 mm, Z = 598.9 mm,       W = 0.5 deg, P = 0.6 deg,
    GP2:
        UF : 1, UT : 2,
       J1 = 0.0 deg, J2 = 0.0 deg
 };
P[220] {
    GP1:
        UF : 6, UT : 5,     CONFIG: 'N U T, 0, 0, 0',
       X = -441.8 mm, Y = 528.9 mm, Z = 598.9 mm,
       W = 0.5 deg, P = 0.5 deg,
    GP2:
        UF : 1, UT : 2,
       J1 = 0.0 deg, J2 = 0.0 deg
 };
P[465] {
    GP1:
        UF : 6, UT : 5,     CONFIG: 'N U T, 0, 0, 0',
 X = -424.8 mm, Y = 599.9 mm, Z = 598.9 mm,       W = 0.5 deg, P = 0.5 deg,
    GP2:
        UF : 1, UT : 2,
       J1 = 0.0 deg, J2 = 0.0 deg
 };
P[221] {
    GP1:
        UF : 6, UT : 5,     CONFIG: 'N U T, 0, 0, 0',
       X = -443.4 mm, Y = 530.3 mm, Z = 598.9 mm,
       W = 0.4 deg, P = 0.5 deg,
    GP2:
        UF : 1, UT : 2,
       J1 = 0.0 deg, J2 = 0.0 deg
 };
P[466] {
    GP1:
        UF : 6, UT : 5,     CONFIG: 'N U T, 0, 0, 0',
 X = -426.4 mm, Y = 601.3 mm, Z = 598.9 mm,       W = 0.4 deg, P = 0.5 deg,
    GP2:
        UF : 1, UT : 2,
       J1 = 0.0 deg, J2 = 0.0 deg
 };
P[222] {
    GP1:
        UF : 6, UT : 5,     CONFIG: 'N U T, 0, 0, 0',
       X = -445.1 mm, Y = 531.9 mm, Z = 598.9 mm,
       W = 0.3 deg, P = 0.4 deg,
    GP2:
        UF : 1, UT : 2,
       J1 = 0.0 deg, J2 = 0.0 deg
 };
P[467] {
    GP1:
        UF : 6, UT : 5,     CONFIG: 'N U T, 0, 0, 0',
 X = -428.1 mm, Y = 602.9 mm, Z = 598.9 mm,       W = 0.3 deg, P = 0.4 deg,
    GP2:
        UF : 1, UT : 2,
       J1 = 0.0 deg, J2 = 0.0 deg
 };
P[223] {
    GP1:
        UF : 6, UT : 5,     CONFIG: 'N U T, 0, 0, 0',
       X = -446.2 mm, Y = 533.6 mm, Z = 598.9 mm,
       W = 0.3 deg, P = 0.4 deg,
    GP2:
        UF : 1, UT : 2,
       J1 = 0.0 deg, J2 = 0.0 deg
 };
P[468] {
    GP1:
        UF : 6, UT : 5,     CONFIG: 'N U T, 0, 0, 0',
 X = -429.2 mm, Y = 604.6 mm, Z = 598.9 mm,       W = 0.3 deg, P = 0.4 deg,
    GP2:
        UF : 1, UT : 2,
       J1 = 0.0 deg, J2 = 0.0 deg
 };
P[224] {
    GP1:
        UF : 6, UT : 5,     CONFIG: 'N U T, 0, 0, 0',
       X = -451.4 mm, Y = 542.1 mm, Z = 598.9 mm,
       W = 0.1 deg, P = 0.2 deg,
    GP2:
        UF : 1, UT : 2,
       J1 = 0.0 deg, J2 = 0.0 deg
 };
P[469] {
    GP1:
        UF : 6, UT : 5,     CONFIG: 'N U T, 0, 0, 0',
 X = -434.4 mm, Y = 613.1 mm, Z = 598.9 mm,       W = 0.1 deg, P = 0.2 deg,
    GP2:
        UF : 1, UT : 2,
       J1 = 0.0 deg, J2 = 0.0 deg
 };
P[225] {
    GP1:
        UF : 6, UT : 5,     CONFIG: 'N U T, 0, 0, 0',
       X = -456.5 mm, Y = 550.7 mm, Z = 598.9 mm,
       W = 0.0 deg, P = 0.0 deg,
    GP2:
        UF : 1, UT : 2,
       J1 = 0.0 deg, J2 = 0.0 deg
 };
P[470] {
    GP1:
        UF : 6, UT : 5,     CONFIG: 'N U T, 0, 0, 0',
 X = -439.5 mm, Y = 621.7 mm, Z = 598.9 mm,       W = 0.0 deg, P = 0.0 deg,
    GP2:
        UF : 1, UT : 2,
       J1 = 0.0 deg, J2 = 0.0 deg
 };
P[226] {
    GP1:
        UF : 6, UT : 5,     CONFIG: 'N U T, 0, 0, 0',
       X = -457.7 mm, Y = 552.8 mm, Z = 598.9 mm,
       W = 0.0 deg, P = 0.0 deg,
    GP2:
        UF : 1, UT : 2,
       J1 = 0.0 deg, J2 = 0.0 deg
 };
P[471] {
    GP1:
        UF : 6, UT : 5,     CONFIG: 'N U T, 0, 0, 0',
 X = -440.7 mm, Y = 623.8 mm, Z = 598.9 mm,       W = 0.0 deg, P = 0.0 deg,
    GP2:
        UF : 1, UT : 2,
       J1 = 0.0 deg, J2 = 0.0 deg
 };
P[227] {
    GP1:
        UF : 6, UT : 5,     CONFIG: 'N U T, 0, 0, 0',
       X = -458.1 mm, Y = 554.3 mm, Z = 598.9 mm,
       W = 0.0 deg, P = 0.0 deg,
    GP2:
        UF : 1, UT : 2,
       J1 = 0.0 deg, J2 = 0.0 deg
 };
P[472] {
    GP1:
        UF : 6, UT : 5,     CONFIG: 'N U T, 0, 0, 0',
 X = -441.1 mm, Y = 625.3 mm, Z = 598.9 mm,       W = 0.0 deg, P = 0.0 deg,
    GP2:
        UF : 1, UT : 2,
       J1 = 0.0 deg, J2 = 0.0 deg
 };
P[228] {
    GP1:
        UF : 6, UT : 5,     CONFIG: 'N U T, 0, 0, 0',
       X = -458.3 mm, Y = 555.2 mm, Z = 598.9 mm,
       W = 0.0 deg, P = 0.0 deg,
    GP2:
        UF : 1, UT : 2,
       J1 = 0.0 deg, J2 = 0.0 deg
 };
P[473] {
    GP1:
        UF : 6, UT : 5,     CONFIG: 'N U T, 0, 0, 0',
 X = -441.3 mm, Y = 626.2 mm, Z = 598.9 mm,       W = 0.0 deg, P = 0.0 deg,
    GP2:
        UF : 1, UT : 2,
       J1 = 0.0 deg, J2 = 0.0 deg
 };
P[229] {
    GP1:
        UF : 6, UT : 5,     CONFIG: 'N U T, 0, 0, 0',
       X = -458.3 mm, Y = 556.1 mm, Z = 598.9 mm,
       W = 0.0 deg, P = 0.0 deg,
    GP2:
        UF : 1, UT : 2,
       J1 = 0.0 deg, J2 = 0.0 deg
 };
P[474] {
    GP1:
        UF : 6, UT : 5,     CONFIG: 'N U T, 0, 0, 0',
 X = -441.3 mm, Y = 627.1 mm, Z = 598.9 mm,       W = 0.0 deg, P = 0.0 deg,
    GP2:
        UF : 1, UT : 2,
       J1 = 0.0 deg, J2 = 0.0 deg
 };
P[230] {
    GP1:
        UF : 6, UT : 5,     CONFIG: 'N U T, 0, 0, 0',
       X = -458.2 mm, Y = 557.0 mm, Z = 598.9 mm,
       W = 0.0 deg, P = 0.0 deg,
    GP2:
        UF : 1, UT : 2,
       J1 = 0.0 deg, J2 = 0.0 deg
 };
P[475] {
    GP1:
        UF : 6, UT : 5,     CONFIG: 'N U T, 0, 0, 0',
 X = -441.2 mm, Y = 628.0 mm, Z = 598.9 mm,       W = 0.0 deg, P = 0.0 deg,
    GP2:
        UF : 1, UT : 2,
       J1 = 0.0 deg, J2 = 0.0 deg
 };
P[231] {
    GP1:
        UF : 6, UT : 5,     CONFIG: 'N U T, 0, 0, 0',
       X = -457.8 mm, Y = 558.8 mm, Z = 598.9 mm,
       W = 0.0 deg, P = 0.0 deg,
    GP2:
        UF : 1, UT : 2,
       J1 = 0.0 deg, J2 = 0.0 deg
 };
P[476] {
    GP1:
        UF : 6, UT : 5,     CONFIG: 'N U T, 0, 0, 0',
 X = -440.8 mm, Y = 629.8 mm, Z = 598.9 mm,       W = 0.0 deg, P = 0.0 deg,
    GP2:
        UF : 1, UT : 2,
       J1 = 0.0 deg, J2 = 0.0 deg
 };
P[232] {
    GP1:
        UF : 6, UT : 5,     CONFIG: 'N U T, 0, 0, 0',
       X = -457.0 mm, Y = 560.3 mm, Z = 598.9 mm,
       W = 0.0 deg, P = 0.0 deg,
    GP2:
        UF : 1, UT : 2,
       J1 = 0.0 deg, J2 = 0.0 deg
 };
P[477] {
    GP1:
        UF : 6, UT : 5,     CONFIG: 'N U T, 0, 0, 0',
 X = -440.0 mm, Y = 631.3 mm, Z = 598.9 mm,       W = 0.0 deg, P = 0.0 deg,
    GP2:
        UF : 1, UT : 2,
       J1 = 0.0 deg, J2 = 0.0 deg
 };
P[233] {
    GP1:
        UF : 6, UT : 5,     CONFIG: 'N U T, 0, 0, 0',
       X = -455.9 mm, Y = 561.7 mm, Z = 598.9 mm,
       W = 0.0 deg, P = 0.0 deg,
    GP2:
        UF : 1, UT : 2,
       J1 = 0.0 deg, J2 = 0.0 deg
 };
P[478] {
    GP1:
        UF : 6, UT : 5,     CONFIG: 'N U T, 0, 0, 0',
 X = -438.9 mm, Y = 632.7 mm, Z = 598.9 mm,       W = 0.0 deg, P = 0.0 deg,
    GP2:
        UF : 1, UT : 2,
       J1 = 0.0 deg, J2 = 0.0 deg
 };
P[234] {
    GP1:
        UF : 6, UT : 5,     CONFIG: 'N U T, 0, 0, 0',
       X = -454.5 mm, Y = 562.8 mm, Z = 598.9 mm,
       W = 0.0 deg, P = 0.0 deg,
    GP2:
        UF : 1, UT : 2,
       J1 = 0.0 deg, J2 = 0.0 deg
 };
P[479] {
    GP1:
        UF : 6, UT : 5,     CONFIG: 'N U T, 0, 0, 0',
 X = -437.5 mm, Y = 633.8 mm, Z = 598.9 mm,       W = 0.0 deg, P = 0.0 deg,
    GP2:
        UF : 1, UT : 2,
       J1 = 0.0 deg, J2 = 0.0 deg
 };
P[235] {
    GP1:
        UF : 6, UT : 5,     CONFIG: 'N U T, 0, 0, 0',
       X = -446.5 mm, Y = 568.0 mm, Z = 598.9 mm,
       W = 0.0 deg, P = 0.0 deg,
    GP2:
        UF : 1, UT : 2,
       J1 = 0.0 deg, J2 = 0.0 deg
 };
P[480] {
    GP1:
        UF : 6, UT : 5,     CONFIG: 'N U T, 0, 0, 0',
 X = -429.5 mm, Y = 639.0 mm, Z = 598.9 mm,       W = 0.0 deg, P = 0.0 deg,
    GP2:
        UF : 1, UT : 2,
       J1 = 0.0 deg, J2 = 0.0 deg
 };
P[236] {
    GP1:
        UF : 6, UT : 5,     CONFIG: 'N U T, 0, 0, 0',
       X = -438.5 mm, Y = 573.2 mm, Z = 598.9 mm,
       W = 0.0 deg, P = 0.0 deg,
    GP2:
        UF : 1, UT : 2,
       J1 = 0.0 deg, J2 = 0.0 deg
 };
P[481] {
    GP1:
        UF : 6, UT : 5,     CONFIG: 'N U T, 0, 0, 0',
 X = -421.5 mm, Y = 644.2 mm, Z = 598.9 mm,       W = 0.0 deg, P = 0.0 deg,
    GP2:
        UF : 1, UT : 2,
       J1 = 0.0 deg, J2 = 0.0 deg
 };
P[237] {
    GP1:
        UF : 6, UT : 5,     CONFIG: 'N U T, 0, 0, 0',
       X = -430.5 mm, Y = 578.4 mm, Z = 598.9 mm,
       W = 0.0 deg, P = 0.0 deg,
    GP2:
        UF : 1, UT : 2,
       J1 = 0.0 deg, J2 = 0.0 deg
 };
P[482] {
    GP1:
        UF : 6, UT : 5,     CONFIG: 'N U T, 0, 0, 0',
 X = -413.5 mm, Y = 649.4 mm, Z = 598.9 mm,       W = 0.0 deg, P = 0.0 deg,
    GP2:
        UF : 1, UT : 2,
       J1 = 0.0 deg, J2 = 0.0 deg
 };
P[238] {
    GP1:
        UF : 6, UT : 5,     CONFIG: 'N U T, 0, 0, 0',
       X = -422.5 mm, Y = 583.6 mm, Z = 598.9 mm,
       W = 0.0 deg, P = 0.0 deg,
    GP2:
        UF : 1, UT : 2,
       J1 = 0.0 deg, J2 = 0.0 deg
 };
P[483] {
    GP1:
        UF : 6, UT : 5,     CONFIG: 'N U T, 0, 0, 0',
 X = -405.5 mm, Y = 654.6 mm, Z = 598.9 mm,       W = 0.0 deg, P = 0.0 deg,
    GP2:
        UF : 1, UT : 2,
       J1 = 0.0 deg, J2 = 0.0 deg
 };
P[239] {
    GP1:
        UF : 6, UT : 5,     CONFIG: 'N U T, 0, 0, 0',
       X = -414.5 mm, Y = 588.8 mm, Z = 598.9 mm,
       W = 0.0 deg, P = 0.0 deg,
    GP2:
        UF : 1, UT : 2,
       J1 = 0.0 deg, J2 = 0.0 deg
 };
P[484] {
    GP1:
        UF : 6, UT : 5,     CONFIG: 'N U T, 0, 0, 0',
 X = -397.5 mm, Y = 659.8 mm, Z = 598.9 mm,       W = 0.0 deg, P = 0.0 deg,
    GP2:
        UF : 1, UT : 2,
       J1 = 0.0 deg, J2 = 0.0 deg
 };
P[240] {
    GP1:
        UF : 6, UT : 5,     CONFIG: 'N U T, 0, 0, 0',
       X = -406.5 mm, Y = 594.0 mm, Z = 598.9 mm,
       W = 0.0 deg, P = 0.0 deg,
    GP2:
        UF : 1, UT : 2,
       J1 = 0.0 deg, J2 = 0.0 deg
 };
P[485] {
    GP1:
        UF : 6, UT : 5,     CONFIG: 'N U T, 0, 0, 0',
 X = -389.5 mm, Y = 665.0 mm, Z = 598.9 mm,       W = 0.0 deg, P = 0.0 deg,
    GP2:
        UF : 1, UT : 2,
       J1 = 0.0 deg, J2 = 0.0 deg
 };
P[241] {
    GP1:
        UF : 6, UT : 5,     CONFIG: 'N U T, 0, 0, 0',
       X = -398.5 mm, Y = 599.2 mm, Z = 598.9 mm,
       W = 0.0 deg, P = 0.0 deg,
    GP2:
        UF : 1, UT : 2,
       J1 = 0.0 deg, J2 = 0.0 deg
 };
P[486] {
    GP1:
        UF : 6, UT : 5,     CONFIG: 'N U T, 0, 0, 0',
 X = -381.5 mm, Y = 670.2 mm, Z = 598.9 mm,       W = 0.0 deg, P = 0.0 deg,
    GP2:
        UF : 1, UT : 2,
       J1 = 0.0 deg, J2 = 0.0 deg
 };
P[242] {
    GP1:
        UF : 6, UT : 5,     CONFIG: 'N U T, 0, 0, 0',
       X = -390.5 mm, Y = 604.4 mm, Z = 598.9 mm,
       W = 0.0 deg, P = 0.0 deg,
    GP2:
        UF : 1, UT : 2,
       J1 = 0.0 deg, J2 = 0.0 deg
 };
P[487] {
    GP1:
        UF : 6, UT : 5,     CONFIG: 'N U T, 0, 0, 0',
 X = -373.5 mm, Y = 675.4 mm, Z = 598.9 mm,       W = 0.0 deg, P = 0.0 deg,
    GP2:
        UF : 1, UT : 2,
       J1 = 0.0 deg, J2 = 0.0 deg
 };
P[243] {
    GP1:
        UF : 6, UT : 5,     CONFIG: 'N U T, 0, 0, 0',
       X = -382.5 mm, Y = 609.6 mm, Z = 598.9 mm,
       W = 0.0 deg, P = 0.0 deg,
    GP2:
        UF : 1, UT : 2,
       J1 = 0.0 deg, J2 = 0.0 deg
 };
P[488] {
    GP1:
        UF : 6, UT : 5,     CONFIG: 'N U T, 0, 0, 0',
 X = -365.5 mm, Y = 680.6 mm, Z = 598.9 mm,       W = 0.0 deg, P = 0.0 deg,
    GP2:
        UF : 1, UT : 2,
       J1 = 0.0 deg, J2 = 0.0 deg
 };
/END
